// TIA Portal V18 export
VAR_GLOBAL   // PLC tag table "AI"
   ina_InductiveResult AT %IW2 : Int;
   ina_1 AT %IW4 : Int;
   in_BaseAxis AT %IW7 : Int;
   ina_Arm1Axis AT %IW10 : Int;
   ina_Arm2Axis AT %IW12 : Int;
   ina_Arm3Axis AT %IW14 : Int;
   ina_ToolAxis AT %IW16 : Int;
   ina_7 AT %IW18 : Int;
   ina_8 AT %IW20 : Int;
   ina_9 AT %IW22 : Int;
   ina_HorizontalAxis AT %IW26 : Int;
   ina_VerticalAxis AT %IW28 : Int;
END_VAR
